% RSLogix 500 project I2P-Job9-Adam Boczkiewicz.RSS, saved by version 10.00.00.00 %
PROJECT "ML04A"    % processor: Bul.1763 MicroLogix 1100 Series B %

PROGRAM FILES
  LAD 2   4 rungs

DATA FILES
  O0 OUTPUT  4 elements
  I1 INPUT  6 elements
  S2 STATUS  66 elements
  B3 BINARY  1 elements
  T4 TIMER  1 elements
  C5 COUNTER  1 elements
  R6 CONTROL  1 elements
  N7 INTEGER  1 elements
  F8 FLOAT  1 elements

LADDER 2
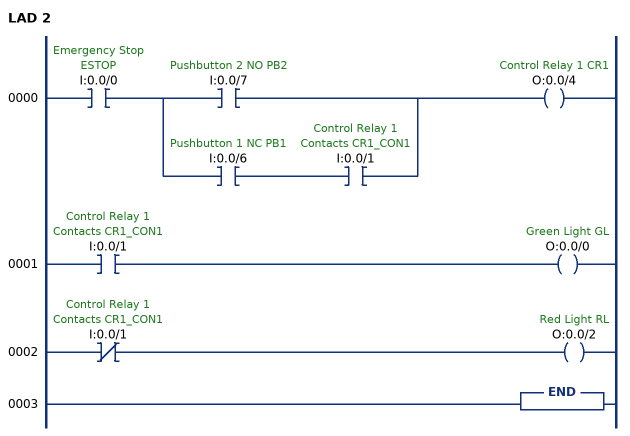
% Rung: 0 %
SOR XIC I:0.0/0 BST XIC I:0.0/7 NXB XIC I:0.0/6 XIC I:0.0/1 BND OTE O:0.0/4 EOR
%   I:0.0/0  ESTOP  "Emergency Stop" %
%   I:0.0/7  PB2  "Pushbutton 2 NO" %
%   I:0.0/6  PB1  "Pushbutton 1 NC" %
%   I:0.0/1  CR1_CON1  "Control Relay 1 Contacts" %
%   O:0.0/4  CR1  "Control Relay 1" %
% Rung: 1 %
SOR XIC I:0.0/1 OTE O:0.0/0 EOR
%   I:0.0/1  CR1_CON1  "Control Relay 1 Contacts" %
%   O:0.0/0  GL  "Green Light" %
% Rung: 2 %
SOR XIO I:0.0/1 OTE O:0.0/2 EOR
%   I:0.0/1  CR1_CON1  "Control Relay 1 Contacts" %
%   O:0.0/2  RL  "Red Light" %
% Rung: 3 %
SOR END EOR

OTHER DOCUMENTED ADDRESSES
  I:0.0/2  CR1_CON2  "Control Relay Contacts 2"
  I:0.0/3  3PSS_A  "3Position Selector Switch Position A"
  I:0.0/4  3PSS_B  "3Position Selector Switch Position B"
  I:0.0/5  2PSS  "2 Position Selector Switch"
  I:0.0/8  PB3  "Pushbutton 3 NO"
  O:0.0/1  YL  "Yellow light"
  O:0.0/3  BL  "Blue Light"
  O:0.0/5  CR2  "Control Relay 2"
